# EPICS substitutions: db/Beckhoff_2XXX/ecmcEP2624-0002.substitutions
file "ecmcEcSlave.template"
{
  pattern {}
          {}
}

file "ecmcEL2XXX-chx.template"
{
  pattern {CH_ID, ZNAM,   ONAM,   ZSV,        OSV,        PINI,  DESC                               }
          {1,     "Zero", "One",  "NO_ALARM", "NO_ALARM", 0,     "$(HWTYPE): Binary Output $(CH_ID)"}
          {2,     "Zero", "One",  "NO_ALARM", "NO_ALARM", 0,     "$(HWTYPE): Binary Output $(CH_ID)"}
          {3,     "Zero", "One",  "NO_ALARM", "NO_ALARM", 0,     "$(HWTYPE): Binary Output $(CH_ID)"}
          {4,     "Zero", "One",  "NO_ALARM", "NO_ALARM", 0,     "$(HWTYPE): Binary Output $(CH_ID)"}
}
